{attribute 'qualified_only'}
VAR_GLOBAL
	//Mode selector booleans
	bManualMode 			: BOOL;
	bAutoMode 				: BOOL;
	
	//Time variables
	fSampleTime				: LREAL := 0.002;
	fTimeSinceStart			: LREAL := 0.0;
	
	//Actuator position data
	fStrokeActuatorMain 	AT %I* : LREAL;
	fStrokeActuatorKnuckle 	AT %I* : LREAL;
	fSlewMotorAngle			AT %I* : LREAL;
	fWinchMotorAngleEncoder		AT %I* : LREAL;	
	fWinchAngle				: LREAL;
	fWinchMotorAngleRefDeg	: LREAL;
	
	//Positions from forward kinematics
	fCraneForwardX 			: LREAL;
	fCraneForwardY 			: LREAL;
	fTheta3Forward			: LREAL;
	fTheta4Forward			: LREAL;
	
	//Working parameters crane
	fWireLengthOnCrane		: LREAL;
	fPayloadHeightIni		: LREAL := 0.0;
	fWinchPitchRadiusLayer1 : LREAL := 0.0716;
	fWinchPitchRadiusLayer2 : LREAL := 0.0731;
	fWinchGearRatio 		: LREAL := 32;
	fWinchMotorAngleAbsRef	: LREAL;
	
	//Encoder values 
	fEncoderValue0Turns		: LREAL := 0.0;
	fEncoderValue5Turns		: LREAL := 0.0;
	fEncoderValueLayer2		: LREAL := 23666.0;
	fEncoderValueStartAuto	: LREAL;
	fTooltipYAutoStart		: LREAL;
	fRefPosPayloadAutoStart	: LREAL;
	fWinchMotorAngleRelRef	: LREAL;
	
	

END_VAR

(* stored: Version 1.1.0.1, ProductVersion 3.1.4024.12
   GVL G_MachineControl: Id {81b36d32-4934-4a29-831b-336ae7ff3ebd} *)
